// TIA Portal V17 export
// export: Created 2025-04-11T04:54:25.15688Z, ExportSetting WithDefaults, DisplayName Totally Integrated Automation Portal, DisplayVersion V17, DisplayName TIA Portal Openness, DisplayVersion V17, DisplayName TIA Portal Version Control Interface, DisplayVersion V17, DisplayName SINAMICS Startdrive Advanced, DisplayVersion V17, DisplayName SINAMICS Startdrive G130, G150, S120, S150, SINAMICS MV, S210, DisplayVersion V17, DisplayName SINAMICS Startdrive G110M, G120, G120C, G120D, G120P, G115D, DisplayVersion V17, DisplayName STEP 7 Professional, DisplayVersion V17, DisplayName STEP 7 Safety, DisplayVersion V17, DisplayName WinCC Advanced, DisplayVersion V17
TYPE "UDT_Ana_ALM"
// stored: IsFailsafeCompliant false
   STRUCT
      OUT_wInterlock : Word;   // 联锁字 (Bit0=高高报警, Bit1=低低报警, Bit2=传感器1故障, Bit3=传感器2故障, Bit4=传感器3故障)
      OUT_LLAlarm : Bool;   // 低低报警
      OUT_HHAlarm : Bool;   // 高高报警
      OUT_SensorFault1 : Bool;   // 传感器1故障
      OUT_SensorFault2 : Bool;   // 传感器2故障
      OUT_SensorFault3 : Bool;   // 传感器3故障
   END_STRUCT;
END_TYPE
